FUNCTION CallHardwareModules : BOOL

robotLeft();
robotRight();

skidLeft();
skidRight();

stagingTableLeft();
stagingTableRight();

skidLeft();
skidRight();

magazineLeft();
magazineRight();

stagingTableLeft();
stagingTableRight();

strapper();

insertionLeft();
insertionRight();
insertionBottom();

stagingTemplateLeft();
stagingTemplateRight();

END_FUNCTION

(* stored: Version 1.1.0.1, ProductVersion 3.1.4024.11
   POU CallHardwareModules: Id {d53bfde7-ef31-4033-a59e-17a8585cdf25}, SpecialFunc None *)
